ABB RAPID module: MainModule.mod

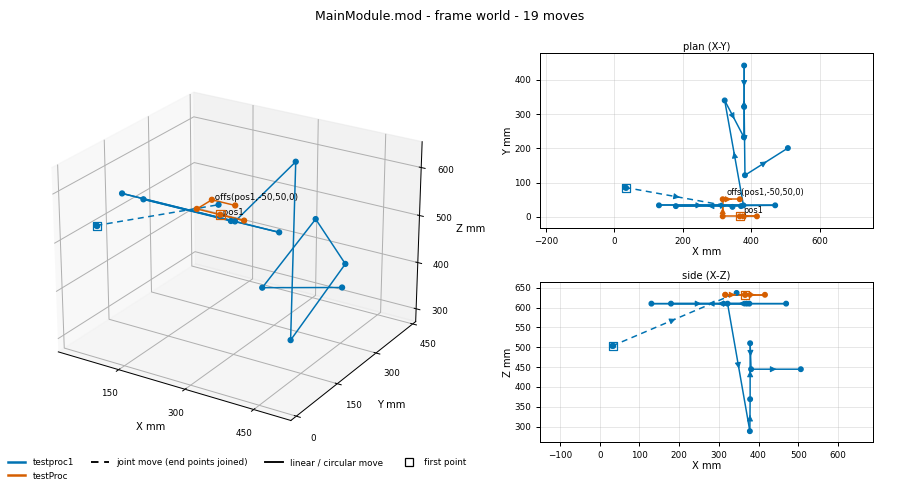
[picture p0: tool path of MainModule.mod in frame world, 19 of 23 moves have a stored position in this frame; points joined in program order, loops and branches not executed]
MODULE MainModule
    CONST jointtarget JtHome:=[[0,0,0,90,0,0],[9E+09,9E+09,9E+09,9E+09,0,9E+09]];
    CONST jointtarget JtCalpos:=[[0,0,0,0,0,0],[9E+09,9E+09,9E+09,9E+09,0,9E+09]];
    CONST jointtarget jtpos1:=[[0,0,0,0,0,0],[9E+09,9E+09,9E+09,9E+09,0,9E+09]];
    CONST robtarget pos1:=[[366.18,1.37,632.09],[0.674845,-0.0204665,0.737511,-0.015567],[0,0,-1,0],[9E+09,9E+09,9E+09,9E+09,9E+09,9E+09]];
	PROC main()
        testProc;
        !moveHome;
       !MoveAbsJ [[0.163419,-71.7784,57.9082,1.86368,14.0725,-4.57856],[9E+09,9E+09,9E+09,9E+09,9E+09,9E+09]]\NoEOffs, v200, z50, tool0;

        !MoveAbsJ[[0,0,0,0,0,0],[9E9,9E9,9E9,9E9,9E9,9E9]];

	ENDPROC





    PROC testproc1( )
        MoveAbsJ [[0.163419,-71.7784,57.9082,1.86368,14.0725,-4.57856],[9E+09,9E+09,9E+09,9E+09,9E+09,9E+09]]\NoEOffs, v1000, z50, tool0;
		MoveJ [[34.10,84.33,503.31],[0.602119,-0.427828,0.569026,0.361422],[0,-1,-1,0],[9E+09,9E+09,9E+09,9E+09,9E+09,9E+09]], v1000, z50, tool0;
		MoveJ [[31.11,85.86,503.15],[0.594905,-0.438541,0.561565,0.372042],[0,-1,-1,0],[9E+09,9E+09,9E+09,9E+09,9E+09,9E+09]], v1000, z50, tool0;
		MoveJ [[344.75,29.07,636.74],[0.641519,-0.0705948,0.763806,-0.00834901],[0,-1,-1,0],[9E+09,9E+09,9E+09,9E+09,9E+09,9E+09]], v1000, z50, tool0;
		MoveAbsJ [[4.89276,-0.257363,0.66943,-1.44968,14.075,-4.5567],[9E+09,9E+09,9E+09,9E+09,9E+09,9E+09]]\NoEOffs, v1000, z50, tool0;
		MoveL [[369.68,31.20,609.82],[0.612284,-0.0729083,0.787227,-0.00815021],[0,-1,-1,0],[9E+09,9E+09,9E+09,9E+09,9E+09,9E+09]], v1000, z50, tool0;
		MoveL [[179.37,31.20,609.81],[0.61228,-0.072914,0.787229,-0.00816186],[0,-1,0,0],[9E+09,9E+09,9E+09,9E+09,9E+09,9E+09]], v1000, z50, tool0;
		MoveL [[469.54,33.54,609.80],[0.612286,-0.0729194,0.787224,-0.00817898],[0,0,-1,0],[9E+09,9E+09,9E+09,9E+09,9E+09,9E+09]], v1000, z50, tool0;
		MoveL [[130.03,33.54,609.79],[0.612278,-0.0729229,0.78723,-0.00817176],[0,-1,0,0],[9E+09,9E+09,9E+09,9E+09,9E+09,9E+09]], v1000, z50, tool0;
		MoveL [[376.81,33.54,609.78],[0.612261,-0.072936,0.787242,-0.00818695],[0,-1,-1,0],[9E+09,9E+09,9E+09,9E+09,9E+09,9E+09]], v1000, z50, tool0;
		MoveL [[321.9909,340.06,609.76],[0.61222,-0.07291,0.78728,-0.00823],[0,-1,0,0],[9E+09,9E+09,9E+09,9E+09,9E+09,9E+09]], v1000, fine, tool0;
		MoveL [[378.14,232.51,288.29],[0.612199,-0.0729154,0.787292,-0.0082291],[0,-2,1,0],[9E+09,9E+09,9E+09,9E+09,9E+09,9E+09]], v1000, z50, tool0;
		MoveL [[378.83,442.01,368.9752],[0.61219,-0.07291,0.7873,-0.00826],[0,-2,1,0],[9E+09,9E+09,9E+09,9E+09,9E+09,9E+09]], v1000, z50, tool0;
		MoveL [[378.84,321.0428,509.9605],[0.61218,-0.07292,0.7873,-0.00824],[0,-1,0,0],[9E+09,9E+09,9E+09,9E+09,9E+09,9E+09]], v1000, z50, tool0;
		MoveL [[381.24,121.52,444.54],[0.612149,-0.0729015,0.787332,-0.00823651],[0,-2,1,0],[9E+09,9E+09,9E+09,9E+09,9E+09,9E+09]], v1000, z50, tool0;
		MoveL [[506.61,200.8426,444.52],[0.61212,-0.07293,0.78735,-0.00823],[0,-2,1,0],[9E+09,9E+09,9E+09,9E+09,9E+09,9E+09]], v1000, z50, tool0;
    ENDPROC


    PROC testProc()
    MoveJ pos1,v50,z15,tool0;
    MoveL offs (pos1,50,0,0),v100,fine,tool0;
    MoveL offs (pos1,-50,0,0),v100,fine,tool0;
    MoveL offs (pos1,-50,50,0),v100,fine,tool0;
    MoveL offs (pos1,0,50,0),v100,fine,tool0;
    ENDPROC

    PROC moveCalPos()

     MoveAbsJ JtCalpos, v50,fine,tool0;
     !Taught position using references
     !MoveAbsJ [[0.200554,-1.15538,-0.473149,0.65211,-0.194197,-3.5621],[9E+09,9E+09,9E+09,9E+09,9E+09,9E+09]]\NoEOffs, v200, fine, tool0;

    ENDPROC
    PROC moveHome()

     MoveAbsJ JtHome, v50,fine,tool0;
     !Taught position using references
     !MoveAbsJ [[0.200554,-1.15538,-0.473149,0.65211,-0.194197,-3.5621],[9E+09,9E+09,9E+09,9E+09,9E+09,9E+09]]\NoEOffs, v200, fine, tool0;

    ENDPROC

ENDMODULE
